{attribute 'qualified_only'}
{attribute 'strict'}
TYPE E_States :
(
	eWaiting := 0,
	eHasCoin,
	eProductEjected,
	eCoinEjected
);
END_TYPE

(* stored: Version 1.1.0.1, ProductVersion 3.1.4022.12
   DUT E_States: Id {973e0ccd-2147-4395-9229-d3fc570a0bb4} *)
